// TwinCAT 3 PLC project plc_kfe_rix_vac_fs
// ProgramVersion: 3.1.4023.0
// libraries:
//   LCLS General, * (SLAC)
//   LCLS Vacuum, * (SLAC - LCLS)
//   PMPS, * (SLAC - LCLS)
//   Tc2_Standard, * (Beckhoff Automation GmbH)
//   Tc2_System, * (Beckhoff Automation GmbH)
//   Tc3_Module, * (Beckhoff Automation GmbH)
// project tree:
//   GVLs/ GVL_RIX_VAC_FSV_PMPS.TcGVL, GVL_RIX_VAC_FS_DEVICES.TcGVL
//   / PlcTask.TcTTO
//   POUs/ MAIN.TcPOU, PRG_KFE_RIX_VAC_FS.TcPOU
// (motion and I/O tree: see PLC project plc_kfe_rix_vac)
// real-time tasks:
//   TASK PlcTask: cycle T#10ms, priority 20, ADS port 350
//   TASK FSTask: cycle T#1ms, priority 19, ADS port 352
// variable links:
//   plc_kfe_rix_vac Instance <-> plc_kfe_rix_vac_fs/plc_kfe_rix_vac_fs Instance
//     PlcTask Inputs/GVL_KFE_RIX_VAC.TV1K2_VFS_Interface.i_eVFS_State <-> PlcTask Outputs/GVL_RIX_VAC_FS_DEVICES.fb_TV1K2_VFS_1.q_eVFS_State
//     PlcTask Inputs/GVL_KFE_RIX_VAC.TV1K2_VFS_Interface.i_xMPS_OK <-> PlcTask Outputs/GVL_RIX_VAC_FS_DEVICES.fb_TV1K2_VFS_1.q_xMPS_OK
//     PlcTask Inputs/GVL_KFE_RIX_VAC.TV1K2_VFS_Interface.i_xTrigger <-> PlcTask Outputs/GVL_RIX_VAC_FS_DEVICES.fb_TV1K2_VFS_1.q_xTrigger
//     PlcTask Inputs/GVL_KFE_RIX_VAC.TV1K2_VFS_Interface.i_xVAC_FAULT_OK <-> PlcTask Outputs/GVL_RIX_VAC_FS_DEVICES.fb_TV1K2_VFS_1.q_xVAC_FAULT_OK
//     PlcTask Inputs/GVL_KFE_RIX_VAC.TV1K2_VFS_Interface.i_xVFS_Closed <-> PlcTask Outputs/GVL_RIX_VAC_FS_DEVICES.fb_TV1K2_VFS_1.q_xVFS_Closed
//     PlcTask Inputs/GVL_KFE_RIX_VAC.TV1K2_VFS_Interface.i_xVFS_Open <-> PlcTask Outputs/GVL_RIX_VAC_FS_DEVICES.fb_TV1K2_VFS_1.q_xVFS_Open
//     PlcTask Outputs/GVL_KFE_RIX_VAC.TV1K2_VFS_Interface.q_xCLS_SW <-> PlcTask Inputs/GVL_RIX_VAC_FS_DEVICES.fb_TV1K2_VFS_1.i_xCLS_SW
//     PlcTask Outputs/GVL_KFE_RIX_VAC.TV1K2_VFS_Interface.q_xOPN_SW <-> PlcTask Inputs/GVL_RIX_VAC_FS_DEVICES.fb_TV1K2_VFS_1.i_xOPN_SW
//     PlcTask Outputs/GVL_KFE_RIX_VAC.TV1K2_VFS_Interface.q_xOverrideMode <-> PlcTask Inputs/GVL_RIX_VAC_FS_DEVICES.fb_TV1K2_VFS_1.i_xOverrideMode
//     PlcTask Outputs/GVL_KFE_RIX_VAC.TV1K2_VFS_Interface.q_xOverrideOpen <-> PlcTask Inputs/GVL_RIX_VAC_FS_DEVICES.fb_TV1K2_VFS_1.i_xOverrideOpen
//     PlcTask Outputs/GVL_KFE_RIX_VAC.TV1K2_VFS_Interface.q_xPRESS_OK <-> PlcTask Inputs/GVL_RIX_VAC_FS_DEVICES.fb_TV1K2_VFS_1.i_xPress_OK
//     PlcTask Outputs/GVL_KFE_RIX_VAC.TV1K2_VFS_Interface.q_xVAC_FAULT_Reset <-> PlcTask Inputs/GVL_RIX_VAC_FS_DEVICES.fb_TV1K2_VFS_1.i_xVAC_FAULT_Reset
//     PlcTask Outputs/GVL_KFE_RIX_VAC.TV1K2_VFS_Interface.q_xVetoValveClosed <-> PlcTask Inputs/GVL_RIX_VAC_FS_DEVICES.fb_TV1K2_VFS_1.i_xVetoValveClosed
//     PlcTask Outputs/GVL_KFE_RIX_VAC.TV1K2_VFS_Interface.q_xVetoValveOpenDO <-> PlcTask Inputs/GVL_RIX_VAC_FS_DEVICES.fb_TV1K2_VFS_1.i_xVetoValveOpenDO

CONFIGURATION plc_kfe_rix_vac_fs
    RESOURCE PLC ON TwinCAT3
        TASK PlcTask(INTERVAL := T#1ms, PRIORITY := 19);
        PROGRAM MAIN WITH PlcTask : MAIN;
    END_RESOURCE
END_CONFIGURATION

// ---- GVLs/GVL_RIX_VAC_FSV_PMPS.TcGVL
VAR_GLOBAL
	{attribute 'pytmc' := '
    	pv: PLC:KFE:RIX:VAC:K2:FFO:02
    '}
    {attribute 'TcLinkTo' := '.q_xFastFaultOut:=TIIB[PMPS_FFO (EL2202)]^Channel 2^Output'}
    g_FastFaultOutput2  :	FB_HardwareFFOutput;	//FFO for Fast Shutter Valves upstream of ST1L0_XTES
END_VAR

// ---- GVLs/GVL_RIX_VAC_FS_DEVICES.TcGVL
VAR_GLOBAL
	
	fb_TV1K2_VFS_1 : FB_VFS;
END_VAR

// ---- POUs/MAIN.TcPOU
PROGRAM MAIN
VAR
END_VAR

PRG_KFE_RIX_VAC_FS();

g_FastFaultOutput2.Execute();

END_PROGRAM

// ---- POUs/PRG_KFE_RIX_VAC_FS.TcPOU
PROGRAM PRG_KFE_RIX_VAC_FS
VAR
END_VAR

//Fast Shutter Valve

fb_TV1K2_VFS_1(
	i_xPMPS_OK:= TRUE, 
	i_xExt_OK:= TRUE, 
	i_sDevName:= 'TV1K2:VFS:1',
	io_fbFFHWO:= g_FastFaultOutput2
);
(*FastFaultOuput*)	
g_FastFaultOutput2.Execute(bAutoReset:= TRUE);

END_PROGRAM
